FUNCTION_BLOCK ABSTRACT CyclicBase EXTENDS Object IMPLEMENTS I_Cyclic
VAR
END_VAR

{analysis -2}

METHOD PUBLIC ABSTRACT Cycle : HRESULT
VAR_INPUT
END_VAR
{analysis -2}
END_METHOD

METHOD RegisterWithParent
VAR_INPUT
	Parent	: I_HostObjects;
END_VAR
Parent.RegisterObject(THIS^);
Parent.RegisterCyclic(THIS^);
END_METHOD

END_FUNCTION_BLOCK

(* stored: Version 1.1.0.1
   POU CyclicBase: Id {822a4270-a76d-44ce-8055-ee2099020175}, SpecialFunc None
   Method Cycle: Id {9762b721-7f92-40df-8e44-4acdbac204f1}
   Method RegisterWithParent: Id {dc0a8f8d-1cb0-4102-9ca6-04d94349ff5f} *)
